// TIA Portal V17 export
// export: Created 2024-09-02T12:50:31.2436841Z, ExportSetting WithDefaults, DisplayName Totally Integrated Automation Portal, DisplayVersion V17, DisplayName TIA Portal Openness, DisplayVersion V17, DisplayName TIA Portal Version Control Interface, DisplayVersion V17, DisplayName STEP 7 Professional, DisplayVersion V17, DisplayName STEP 7 Safety, DisplayVersion V17, DisplayName WinCC Professional, DisplayVersion V17
TYPE "UFM_ActiveTaskDescriptor"
TITLE = UFM_ActiveTaskDescriptor
// (Internal usage only)
// stored: IsFailsafeCompliant false
   STRUCT
      TaskId : Word;
      TaskTypeCode : Int;
   END_STRUCT;
END_TYPE
